{attribute 'qualified_only'}
{attribute 'strict'}
TYPE nUnderPressureTestErrorCodes_V2 :
(
	TestTimeOut := 860,
	SafetyError := 861
	
);
END_TYPE

(* stored: Version 1.1.0.1, ProductVersion 3.1.4024.13
   DUT nUnderPressureTestErrorCodes_V2: Id {1af8e9ac-e0c2-410e-aeb7-01bac62342e0} *)
